{attribute 'linkalways'} 
{attribute 'no_explicit_call' := 'This FB is a CLASS and must be accessed using methods or properties'}
{attribute 'enable_dynamic_creation'}
FUNCTION_BLOCK Node_F_VN_ExportContainer_String EXTENDS VisionNode
VAR
    ipContainer : _ITcVnContainer;
    sText : _STRING('');
    nMaxLength : _ULINT(0);
    hrPrev : _HRESULT(S_OK);
	hresult : _HRESULT(S_OK);
END_VAR

METHOD PUBLIC  Clone : I_Node
VAR
	pNode : POINTER TO Node_F_VN_ExportContainer_String;
END_VAR
pNode := __NEW(Node_F_VN_ExportContainer_String);
Clone := pNode^;
END_METHOD

METHOD FB_init : BOOL
VAR_INPUT
	bInitRetains : BOOL; // if TRUE, the retain variables are initialized (warm start / cold start)
	bInCopyCode : BOOL;  // if TRUE, the instance afterwards gets moved into the copy code (online change)
END_VAR
AddInput('ipContainer', ipContainer);
AddParameter('nMaxLength', nMaxLength);
AddInput('hrPrev', hrPrev);
AddOutput('sText', sText);
AddOutput('hresult',hresult);
END_METHOD

METHOD PROTECTED OnExecute
hresult.Value := F_VN_ExportContainer_String(
	ipContainer := ipContainer.Value,
    sText := sText.Value,
    nMaxLength := nMaxLength.Value,
	hrPrev:= hrPrev.Value);
END_METHOD

METHOD PUBLIC PreExecutionCheck
VAR_INPUT
	Check : I_PreExecutionChecks;
END_VAR
Check.IsTrue(ipContainer.IsValid, 'ipContainer must be a valid container');
Check.IsTrue(ipContainer.IsType(TC_GLOBAL_CONST_LIST.ContainerType_String_SINT), 'ipContainer contains incorrect type');
END_METHOD

END_FUNCTION_BLOCK

(* stored: Version 1.1.0.1, ProductVersion 3.1.4026.13
   POU Node_F_VN_ExportContainer_String: Id {fc7954cb-043b-0b29-082e-f9222eef4403}, SpecialFunc None
   Folder Constructor: Id {95887750-1fe0-005d-2b5b-eb9a6e457191}
   Method Clone: Id {245c1157-1bd1-012d-2aa5-d1b96cafe202}
   Method FB_init: Id {05807364-c2cb-02bf-2bf4-ce3bc4438a6d}
   Method OnExecute: Id {20c90129-3780-0722-3b51-725625fd7cb9}
   Method PreExecutionCheck: Id {0ee15540-6373-0dc4-128f-dc9d8100c5aa} *)
